FUNCTION_BLOCK EspObjectUpdater
VAR_INPUT
END_VAR
VAR_OUTPUT
END_VAR
VAR
END_VAR

END_FUNCTION_BLOCK

(* stored: Version 1.1.0.1
   POU EspObjectUpdater: Id {70f11a0c-3775-4d14-a128-5ab536b4467f}, SpecialFunc None *)
